ORGANIZATION_BLOCK PRINCIPAL:OB1
TITLE=COMENTARIOS DEL PROGRAMA
BEGIN
Network 1 // Título de segmento
// Comentario de segmento
LD     SM0.1
S      M0.1, 1
R      M0.2, 1
Network 2
LD     M0.1
A      I0.0
S      M0.2, 1
R      M0.1, 1
Network 3
LD     M0.2
AN     I0.0
S      M0.1, 1
R      M0.2, 1
Network 4
LD     M0.2
=      Q0.0
END_ORGANIZATION_BLOCK
SUBROUTINE_BLOCK SBR_0:SBR0
TITLE=COMENTARIOS DE LA SUBRUTINA
BEGIN
Network 1 // Título de segmento
// Comentario de segmento
END_SUBROUTINE_BLOCK
INTERRUPT_BLOCK INT_0:INT0
TITLE=COMENTARIOS DE LA RUTINA DE INTERRUPCIÓN
BEGIN
Network 1 // Título de segmento
// Comentario de segmento
END_INTERRUPT_BLOCK
